// Mitsubishi GX Works2 project: PLC_FINAL   PLC: FX3G

// global labels: Global1
VAR_GLOBAL
  start_day AT X007 : BOOL;
  work_day AT Y007 : BOOL;
  start_procces AT M0 : BOOL;
  emergency_btn AT X005 : BOOL;
  rasberry_start_day AT D1100 : REAL;
  lemon_start_day AT D1200 : REAL;
  gummy_start_day AT D1400 : REAL;
  stabilizer_start_day AT D1300 : REAL;
  rasberry AT D1102 : REAL;
  rasberry_stock AT D1102 : REAL;
  lemon_stock AT D1202 : REAL;
  stabilizer_stock AT D1302 : REAL;
  gummy_stock AT D1402 : REAL;
  no_stock AT M0 : BOOL;
  finish_pack AT M1 : BOOL;
  choose_type AT X001 : BOOL;
  analog_input1 AT D8280 : INT;
  analog_output AT D8282 : INT;
  iceCream_type AT D1500 : REAL;
END_VAR
VAR_GLOBAL CONSTANT
  five : REAL := 5.0;
  six : REAL := 6.0;
END_VAR
VAR_GLOBAL
  gumigamRAGIL AT M2 : BOOL;
  gumigamPINUK AT M3 : BOOL;
END_VAR
VAR_GLOBAL CONSTANT
  min_rasberry_RAGIL : REAL := 280.0;
  min_lemon_RAGIL : REAL := 455.0;
  min_stabilizer_RAGIL : REAL := 105.0;
  min_gummy_RAGIL : REAL := 28.0;
  min_gummy_PINUK : REAL := 70.0;
  min_stabilizer_PINUK : REAL := 210.0;
  min_rasberry_PINUK : REAL := 385.0;
  min_lemon_PINUK : REAL := 665.0;
END_VAR
VAR_GLOBAL
  making_timer AT TC1 : BOOL;
END_VAR
VAR_GLOBAL CONSTANT
  fiveSEC : INT := 50;
END_VAR
VAR_GLOBAL
  GLIDA_ready AT TS1 : BOOL;
  start_cooling AT X002 : BOOL;
END_VAR
VAR_GLOBAL CONSTANT
  cast_divide : REAL := 404.5;
END_VAR
VAR_GLOBAL
  GLIDA_in_process AT Y000 : BOOL;
  cooling_timer AT TC2 : BOOL;
END_VAR
VAR_GLOBAL CONSTANT
  eightSEC : INT := 80;
END_VAR
VAR_GLOBAL
  is_below10 AT X003 : BOOL;
  cooling_timer_end AT TS2 : BOOL;
  is_cooling AT Y002 : BOOL;
END_VAR
VAR_GLOBAL CONSTANT
  mix_timeRAGIL : INT := 30;
  mix_timePINUK : INT := 50;
END_VAR
VAR_GLOBAL
  mixing_timerRAGIL AT TC3 : BOOL;
  mixing_timerPINUK AT TC4 : BOOL;
  mixing_endRAGIL AT TS3 : BOOL;
  mixing_lamp_timer1 AT TC5 : BOOL;
  blinking_timer1_end AT TS5 : BOOL;
  blinking_timer1 AT TC5 : BOOL;
  blinking_timer1END AT TS5 : BOOL;
  blinking_timer2 AT TC6 : BOOL;
  blinking_timer2END AT TS6 : BOOL;
  mixing_cycle AT M4 : BOOL;
  mixing_lamp1 AT Y005 : BOOL;
  mixing_lamp2 AT Y006 : BOOL;
  mixing_endPINUK AT TS4 : BOOL;
  coolingEND AT M5 : BOOL;
  m_6 AT M6 : BOOL;
  start_packing AT X004 : BOOL;
  pack_unit AT X000 : BOOL;
  is_packing AT Y004 : BOOL;
END_VAR
VAR_GLOBAL CONSTANT
  seven_gumigams : INT := 7;
END_VAR
VAR_GLOBAL
  counter_unitPacked AT CC0 : BOOL;
  gumigam_in_Box AT CN0 : INT;
END_VAR
VAR_GLOBAL CONSTANT
  zero : REAL;
END_VAR
VAR_GLOBAL
  new_box AT M6 : BOOL;
  counter_unitPackedEND AT CS0 : BOOL;
  storage AT D2000 : REAL;
END_VAR
VAR_GLOBAL CONSTANT
  one_box : REAL := 1.0;
  oneSEC : INT := 10;
END_VAR
VAR_GLOBAL
  enough_stock AT M20 : BOOL;
  work_dayEND AT M30 : BOOL;
  check AT Y010 : BOOL;
END_VAR
VAR_GLOBAL CONSTANT
  ten : REAL := 10.0;
  cast_multiply : REAL := 40.0;
END_VAR
VAR_GLOBAL
  storage_output AT D3000 : REAL;
  pulse_stock_CHECK AT Y010 : BOOL;
  no_initial_stock AT M50 : BOOL;
  rasberry_making AT D1600 : REAL;
  lemon_making AT D1602 : REAL;
END_VAR
VAR_GLOBAL CONSTANT
  ras_for_ras_RAGIL : REAL := 280.0;
  lem_for_ras_RAGIL : REAL := 35;
  lem_for_lem_RAGIL : REAL := 420;
  stab_for_ras_RAGIL : REAL := 35;
  stab_for_lem_RAGIL : REAL := 70;
  ras_for_ras_PINUK : REAL := 385;
  lem_for_ras_PINUK : REAL := 105;
  lem_for_lem_PINUK : REAL := 560;
  stab_for_ras_PINUK : REAL := 70;
  stab_for_lem_PINUK : REAL := 140;
END_VAR
VAR_GLOBAL
  iceCream_mixing AT D1800 : REAL;
  rasberry_cooling AT D1700 : REAL;
  lemon_cooling AT D1702 : REAL;
END_VAR
VAR_GLOBAL CONSTANT
  zero_word : INT;
END_VAR

// task Task_01 (event TRUE, interval 0, priority 31): POU_01

PROGRAM POU_01
(* structured ladder/FBD written out as ST: instructions are called as NAME(EN, inputs, outputs); _pN, _eN, _tN stand for wires *)
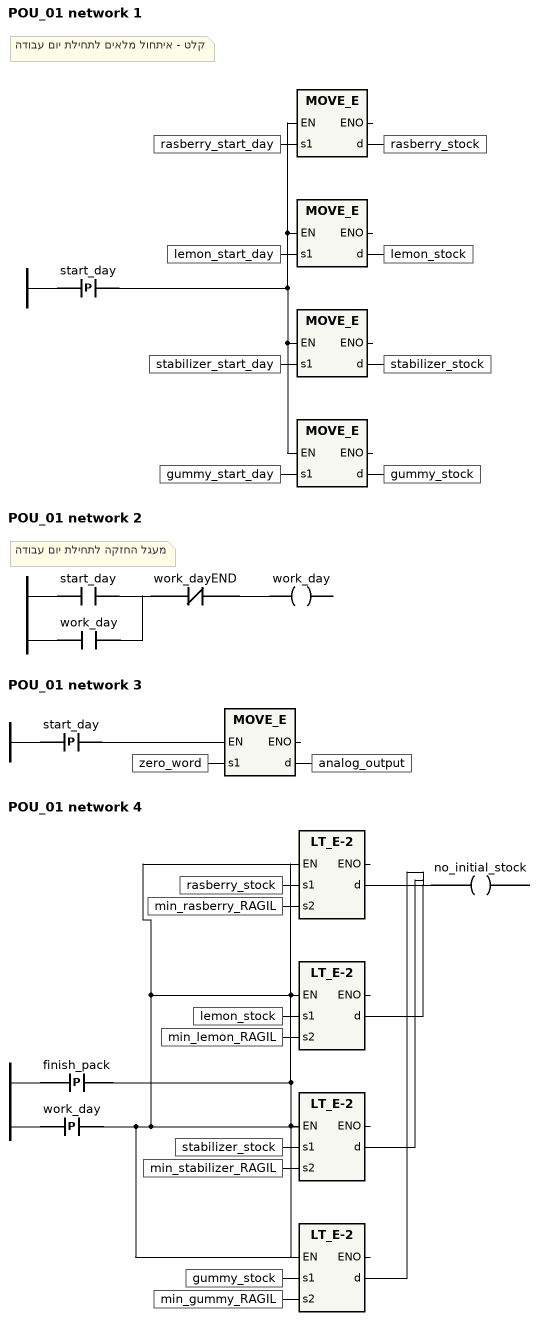
(* network 1 *)
(* קלט - איתחול מלאים לתחילת יום עבודה *)
_p1 := LDP(TRUE, start_day);
MOVE_E(_p1, rasberry_start_day, rasberry_stock);
MOVE_E(_p1, lemon_start_day, lemon_stock);
MOVE_E(_p1, stabilizer_start_day, stabilizer_stock);
MOVE_E(_p1, gummy_start_day, gummy_stock);
(* network 2 *)
(* מעגל החזקה לתחילת יום עבודה *)
work_day := (start_day OR work_day) AND NOT work_dayEND;
(* network 3 *)
MOVE_E(LDP(TRUE, start_day), zero_word, analog_output);
(* network 4 *)
_p1 := LDP(TRUE, finish_pack) OR LDP(TRUE, work_day);
LT_E(_p1, rasberry_stock, min_rasberry_RAGIL, _t2);
LT_E(_p1, lemon_stock, min_lemon_RAGIL, _t3);
LT_E(_p1, stabilizer_stock, min_stabilizer_RAGIL, _t4);
LT_E(_p1, gummy_stock, min_gummy_RAGIL, _t5);
no_initial_stock := _t2 OR _t3 OR _t4 OR _t5;
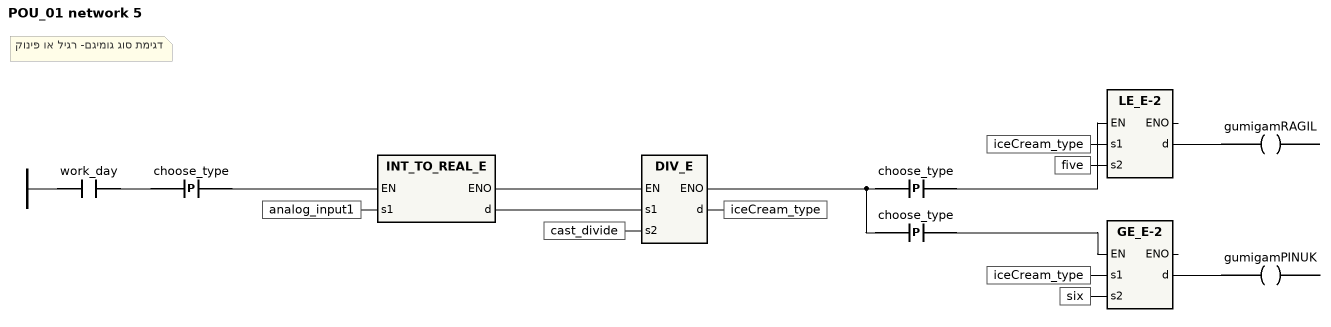
(* network 5 *)
(* דגימת סוג גומיגם- רגיל או פינוק *)
_e2 := INT_TO_REAL_E(work_day AND LDP(TRUE, choose_type), analog_input1, _t1);
_e3 := DIV_E(_e2, _t1, cast_divide, iceCream_type);
LE_E(_e3 AND LDP(TRUE, choose_type), iceCream_type, five, _t4);
gumigamRAGIL := _t4;
GE_E(_e3 AND LDP(TRUE, choose_type), iceCream_type, six, _t5);
gumigamPINUK := _t5;
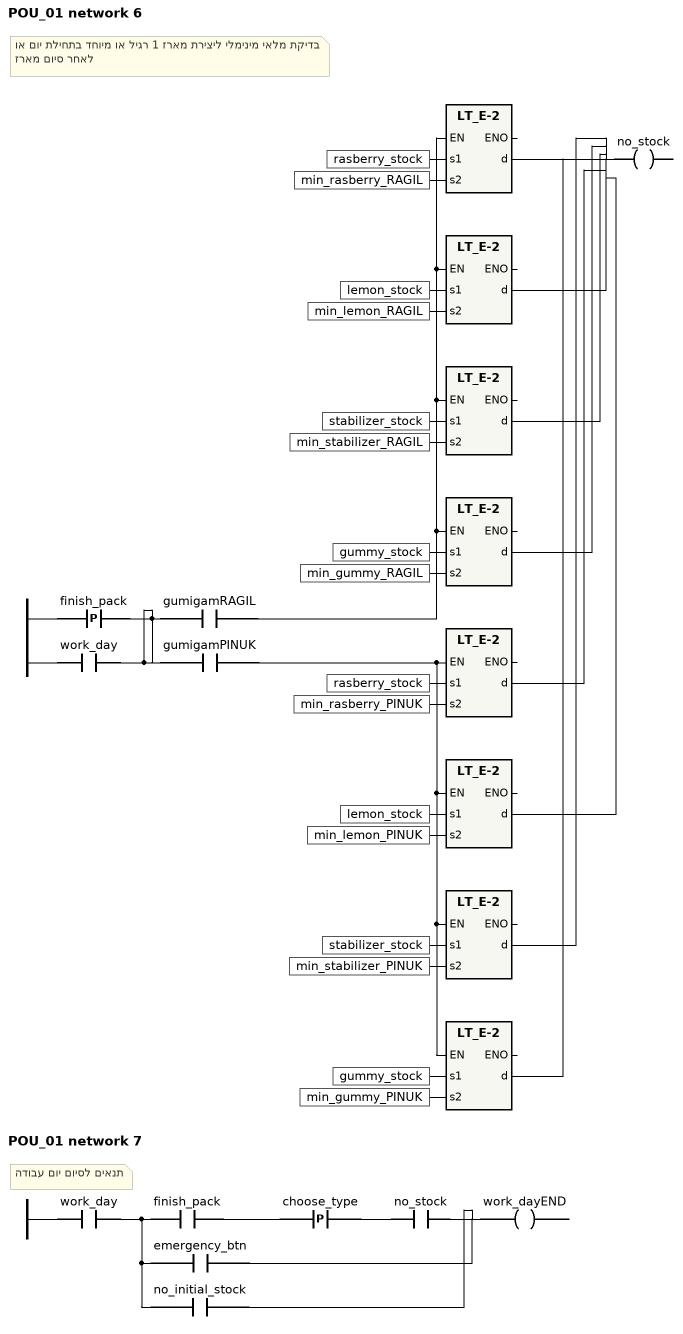
(* network 6 *)
(* בדיקת מלאי מינימלי ליצירת מארז 1 רגיל או מיוחד בתחילת יום או לאחר סיום מארז *)
_p1 := LDP(TRUE, finish_pack) OR work_day;
_p2 := _p1 AND gumigamRAGIL;
LT_E(_p2, rasberry_stock, min_rasberry_RAGIL, _t3);
LT_E(_p2, lemon_stock, min_lemon_RAGIL, _t4);
LT_E(_p2, stabilizer_stock, min_stabilizer_RAGIL, _t5);
LT_E(_p2, gummy_stock, min_gummy_RAGIL, _t6);
_p7 := _p1 AND gumigamPINUK;
LT_E(_p7, rasberry_stock, min_rasberry_PINUK, _t8);
LT_E(_p7, lemon_stock, min_lemon_PINUK, _t9);
LT_E(_p7, stabilizer_stock, min_stabilizer_PINUK, _t10);
LT_E(_p7, gummy_stock, min_gummy_PINUK, _t11);
no_stock := _t3 OR _t4 OR _t5 OR _t6 OR _t8 OR _t9 OR _t10 OR _t11;
(* network 7 *)
(* תנאים לסיום יום עבודה *)
work_dayEND := (work_day AND finish_pack AND LDP(TRUE, choose_type) AND no_stock) OR (work_day AND emergency_btn) OR (work_day AND no_initial_stock);
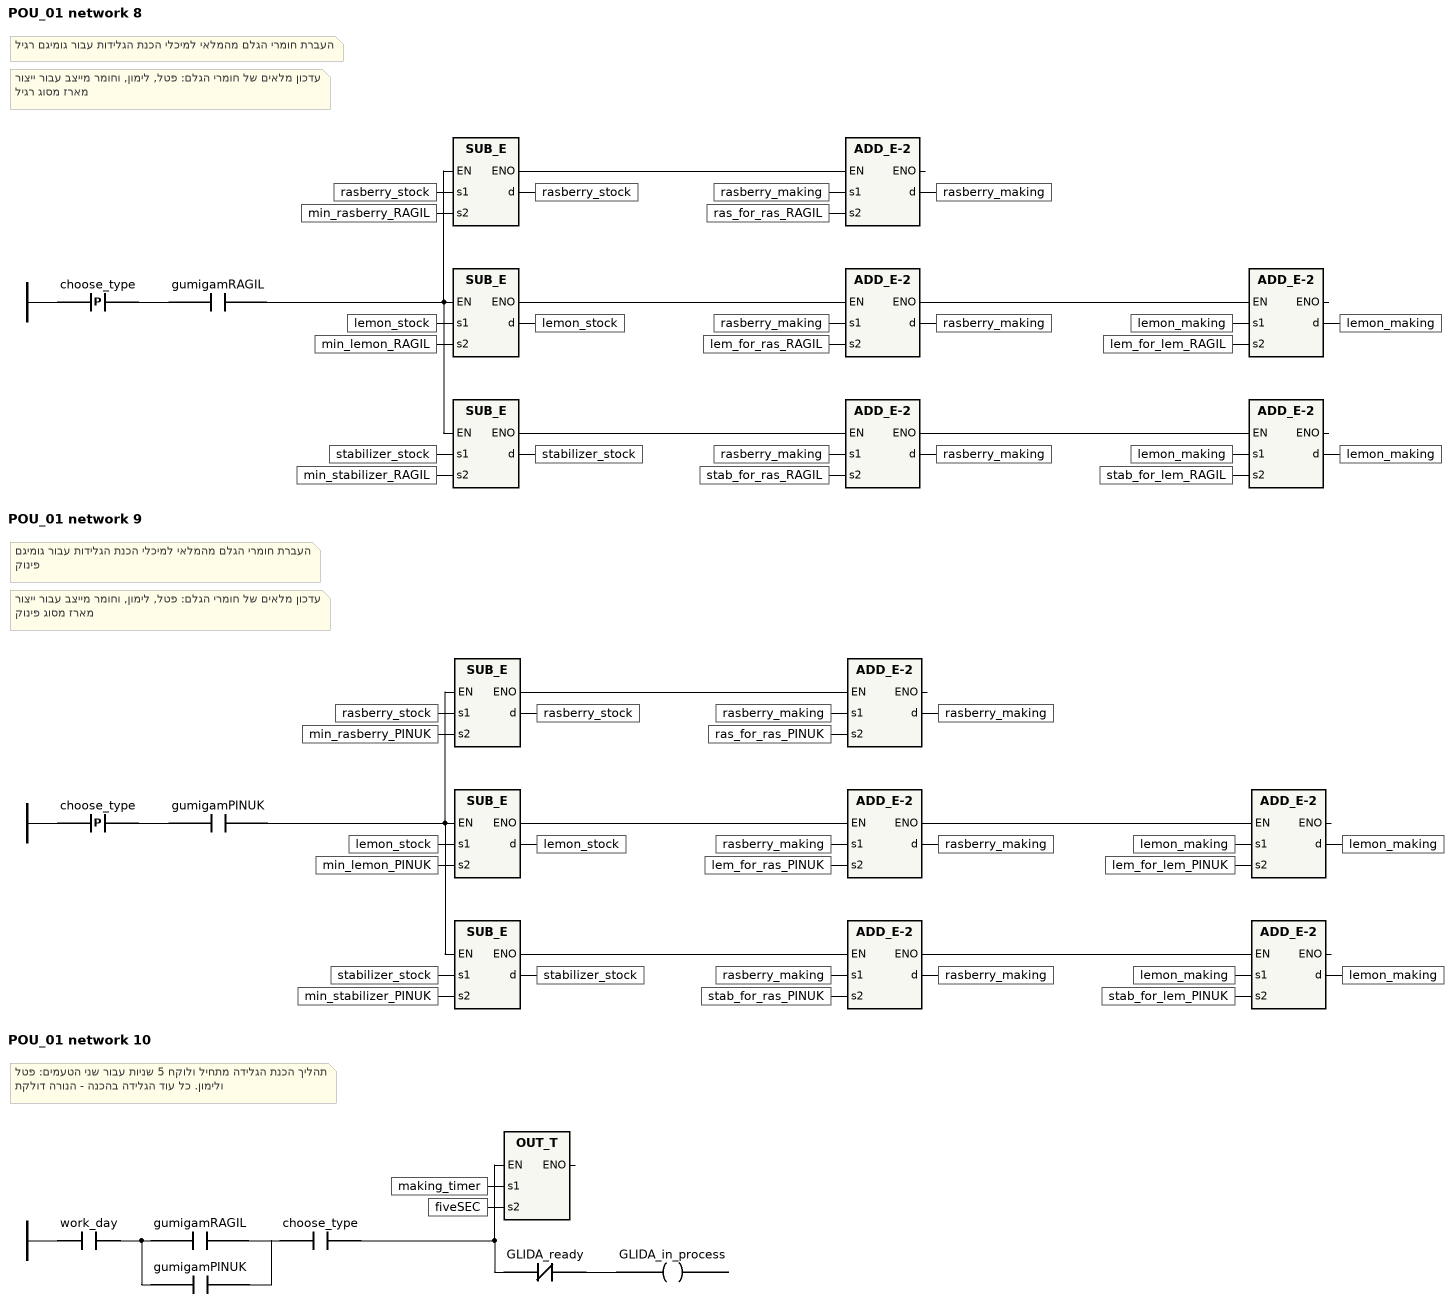
(* network 8 *)
(* העברת חומרי הגלם מהמלאי למיכלי הכנת הגלידות עבור גומיגם רגיל *)
(* עדכון מלאים של חומרי הגלם: פטל, לימון, וחומר מייצב עבור ייצור מארז מסוג רגיל *)
_p1 := LDP(TRUE, choose_type) AND gumigamRAGIL;
_e2 := SUB_E(_p1, rasberry_stock, min_rasberry_RAGIL, rasberry_stock);
ADD_E(_e2, rasberry_making, ras_for_ras_RAGIL, rasberry_making);
_e3 := SUB_E(_p1, lemon_stock, min_lemon_RAGIL, lemon_stock);
_e4 := ADD_E(_e3, rasberry_making, lem_for_ras_RAGIL, rasberry_making);
ADD_E(_e4, lemon_making, lem_for_lem_RAGIL, lemon_making);
_e5 := SUB_E(_p1, stabilizer_stock, min_stabilizer_RAGIL, stabilizer_stock);
_e6 := ADD_E(_e5, rasberry_making, stab_for_ras_RAGIL, rasberry_making);
ADD_E(_e6, lemon_making, stab_for_lem_RAGIL, lemon_making);
(* network 9 *)
(* העברת חומרי הגלם מהמלאי למיכלי הכנת הגלידות עבור גומיגם פינוק *)
(* עדכון מלאים של חומרי הגלם: פטל, לימון, וחומר מייצב עבור ייצור מארז מסוג פינוק *)
_p1 := LDP(TRUE, choose_type) AND gumigamPINUK;
_e2 := SUB_E(_p1, rasberry_stock, min_rasberry_PINUK, rasberry_stock);
ADD_E(_e2, rasberry_making, ras_for_ras_PINUK, rasberry_making);
_e3 := SUB_E(_p1, lemon_stock, min_lemon_PINUK, lemon_stock);
_e4 := ADD_E(_e3, rasberry_making, lem_for_ras_PINUK, rasberry_making);
ADD_E(_e4, lemon_making, lem_for_lem_PINUK, lemon_making);
_e5 := SUB_E(_p1, stabilizer_stock, min_stabilizer_PINUK, stabilizer_stock);
_e6 := ADD_E(_e5, rasberry_making, stab_for_ras_PINUK, rasberry_making);
ADD_E(_e6, lemon_making, stab_for_lem_PINUK, lemon_making);
(* network 10 *)
(* תהליך הכנת הגלידה מתחיל ולוקח 5 שניות עבור שני הטעמים: פטל ולימון. כל עוד הגלידה בהכנה - הנורה דולקת *)
_p1 := ((work_day AND gumigamRAGIL) OR (work_day AND gumigamPINUK)) AND choose_type;
OUT_T(_p1, making_timer, fiveSEC);
GLIDA_in_process := _p1 AND NOT GLIDA_ready;
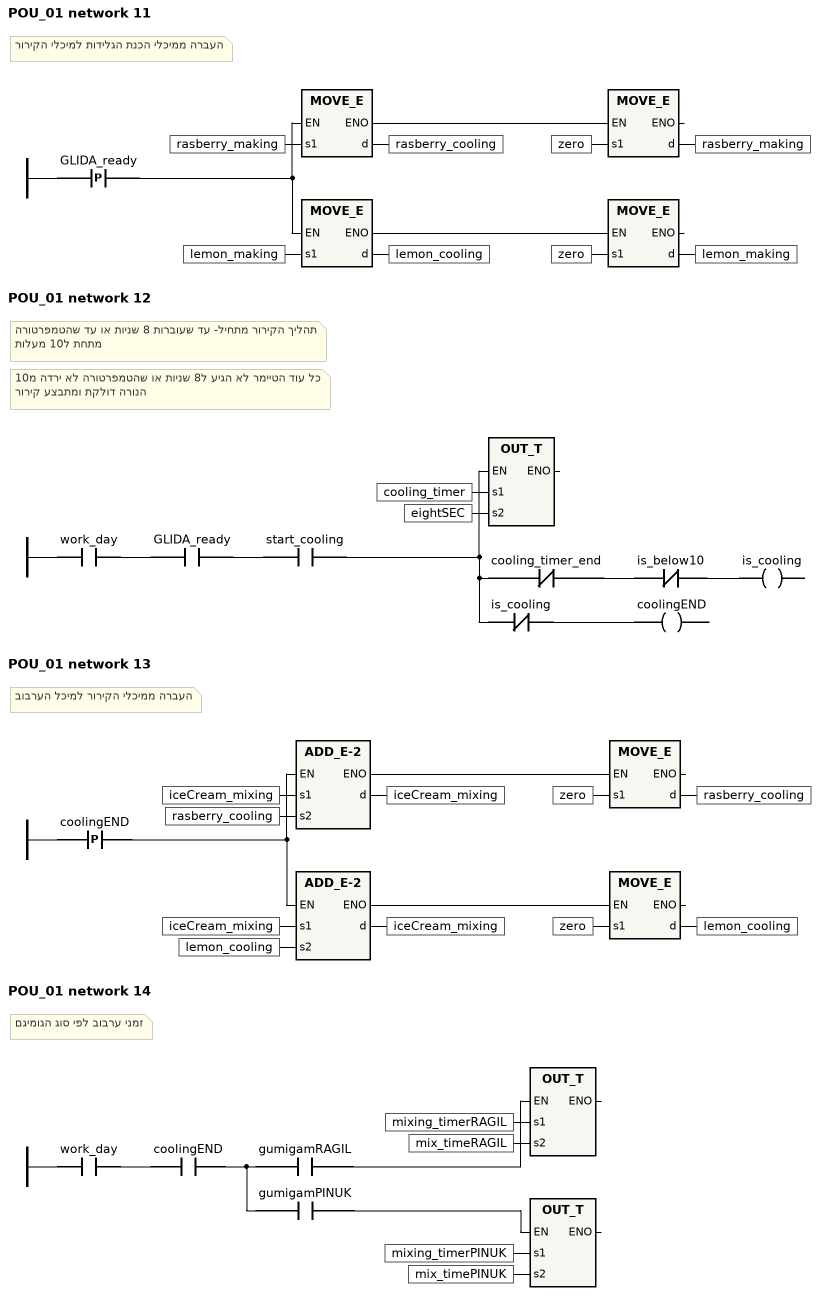
(* network 11 *)
(* העברה ממיכלי הכנת הגלידות למיכלי הקירור *)
_p1 := LDP(TRUE, GLIDA_ready);
_e2 := MOVE_E(_p1, rasberry_making, rasberry_cooling);
MOVE_E(_e2, zero, rasberry_making);
_e3 := MOVE_E(_p1, lemon_making, lemon_cooling);
MOVE_E(_e3, zero, lemon_making);
(* network 12 *)
(* תהליך הקירור מתחיל- עד שעוברות 8 שניות או עד שהטמפרטורה מתחת ל10 מעלות *)
(* כל עוד הטיימר לא הגיע ל8 שניות או שהטמפרטורה לא ירדה מ10 הנורה דולקת ומתבצע קירור *)
_p1 := work_day AND GLIDA_ready AND start_cooling;
OUT_T(_p1, cooling_timer, eightSEC);
is_cooling := _p1 AND NOT cooling_timer_end AND NOT is_below10;
coolingEND := _p1 AND NOT is_cooling;
(* network 13 *)
(* העברה ממיכלי הקירור למיכל הערבוב *)
_p1 := LDP(TRUE, coolingEND);
_e2 := ADD_E(_p1, iceCream_mixing, rasberry_cooling, iceCream_mixing);
MOVE_E(_e2, zero, rasberry_cooling);
_e3 := ADD_E(_p1, iceCream_mixing, lemon_cooling, iceCream_mixing);
MOVE_E(_e3, zero, lemon_cooling);
(* network 14 *)
(* זמני ערבוב לפי סוג הגומיגם *)
_p1 := work_day AND coolingEND;
OUT_T(_p1 AND gumigamRAGIL, mixing_timerRAGIL, mix_timeRAGIL);
OUT_T(_p1 AND gumigamPINUK, mixing_timerPINUK, mix_timePINUK);
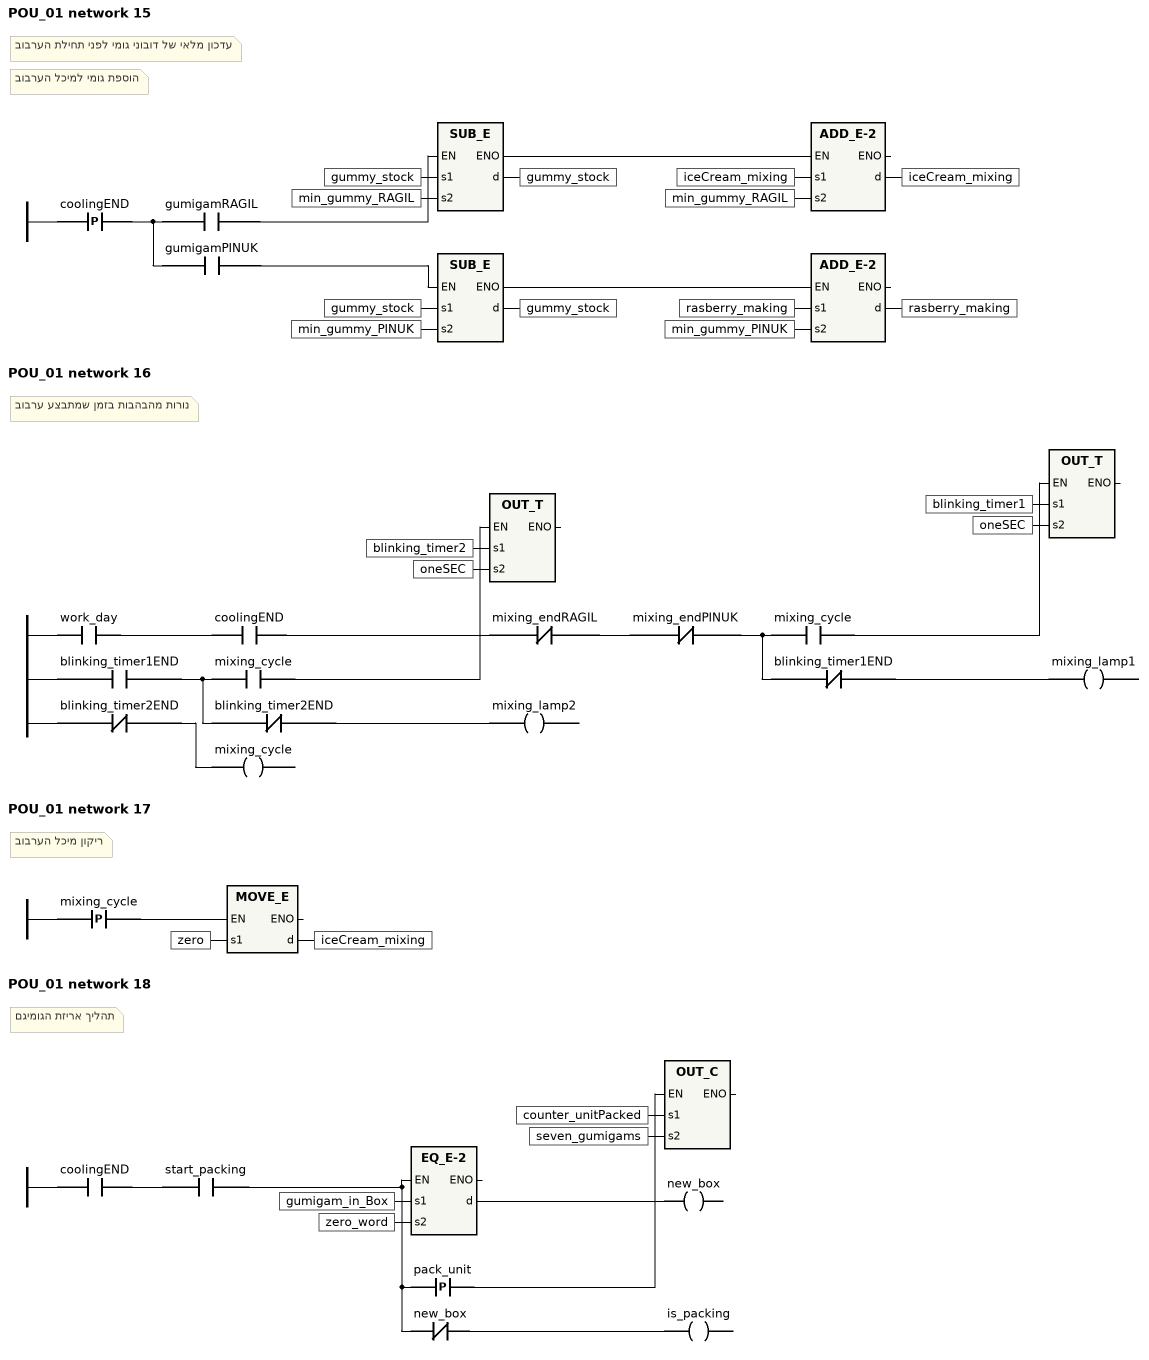
(* network 15 *)
(* עדכון מלאי של דובוני גומי לפני תחילת הערבוב *)
(* הוספת גומי למיכל הערבוב *)
_p1 := LDP(TRUE, coolingEND);
_e2 := SUB_E(_p1 AND gumigamRAGIL, gummy_stock, min_gummy_RAGIL, gummy_stock);
ADD_E(_e2, iceCream_mixing, min_gummy_RAGIL, iceCream_mixing);
_e3 := SUB_E(_p1 AND gumigamPINUK, gummy_stock, min_gummy_PINUK, gummy_stock);
ADD_E(_e3, rasberry_making, min_gummy_PINUK, rasberry_making);
(* network 16 *)
(* נורות מהבהבות בזמן שמתבצע ערבוב *)
_p1 := work_day AND coolingEND AND NOT mixing_endRAGIL AND NOT mixing_endPINUK;
OUT_T(_p1 AND mixing_cycle, blinking_timer1, oneSEC);
mixing_lamp1 := _p1 AND NOT blinking_timer1END;
OUT_T(blinking_timer1END AND mixing_cycle, blinking_timer2, oneSEC);
mixing_lamp2 := blinking_timer1END AND NOT blinking_timer2END;
mixing_cycle := NOT blinking_timer2END;
(* network 17 *)
(* ריקון מיכל הערבוב *)
MOVE_E(LDP(TRUE, mixing_cycle), zero, iceCream_mixing);
(* network 18 *)
(* תהליך אריזת הגומיגם *)
_p1 := coolingEND AND start_packing;
OUT_C(_p1 AND LDP(TRUE, pack_unit), counter_unitPacked, seven_gumigams);
EQ_E(_p1, gumigam_in_Box, zero_word, _t2);
new_box := _t2;
is_packing := _p1 AND NOT new_box;
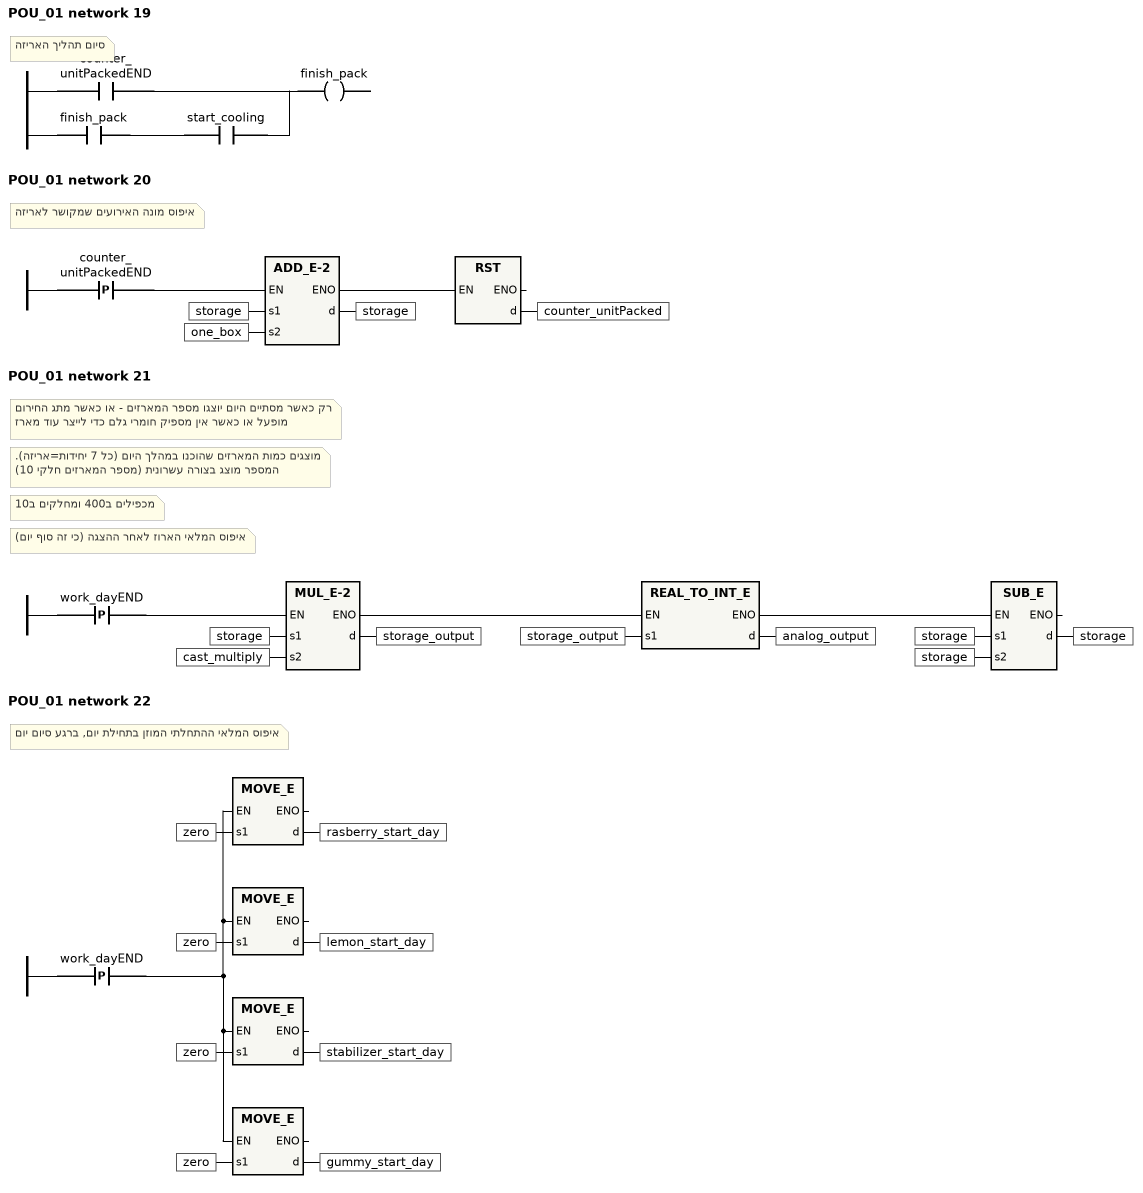
(* network 19 *)
(* סיום תהליך האריזה *)
finish_pack := counter_unitPackedEND OR (finish_pack AND start_cooling);
(* network 20 *)
(* איפוס מונה האירועים שמקושר לאריזה *)
_e1 := ADD_E(LDP(TRUE, counter_unitPackedEND), storage, one_box, storage);
RST(_e1, counter_unitPacked);
(* network 21 *)
(* רק כאשר מסתיים היום יוצגו מספר המארזים - או כאשר מתג החירום מופעל או כאשר אין מספיק חומרי גלם כדי לייצר עוד מארז *)
(* מוצגים כמות המארזים שהוכנו במהלך היום (כל 7 יחידות=אריזה). המספר מוצג בצורה עשרונית (מספר המארזים חלקי 10) *)
(* מכפילים ב400 ומחלקים ב10 *)
(* איפוס המלאי הארוז לאחר ההצגה (כי זה סוף יום) *)
_e1 := MUL_E(LDP(TRUE, work_dayEND), storage, cast_multiply, storage_output);
_e2 := REAL_TO_INT_E(_e1, storage_output, analog_output);
SUB_E(_e2, storage, storage, storage);
(* network 22 *)
(* איפוס המלאי ההתחלתי המוזן בתחילת יום, ברגע סיום יום *)
_p1 := LDP(TRUE, work_dayEND);
MOVE_E(_p1, zero, rasberry_start_day);
MOVE_E(_p1, zero, lemon_start_day);
MOVE_E(_p1, zero, stabilizer_start_day);
MOVE_E(_p1, zero, gummy_start_day);
END_PROGRAM
